Staubli VAL3: getMedian.pgx

public program getMedian(num& x_nInput[], num& x_nMedian)
  local num l_nCount
  local num l_nSmallsub
  local num l_nSort
  local num l_nTemp
begin

  // do a selection sort:
  // The idea of Selection Sort is that we repeatedly find the smallest element in the unsorted part of the array and swap it with the first element in the unsorted part of the array.

  resize(nTemp, 1, size(x_nInput))
  resize(nCopy, 1, size(x_nInput))

  for l_nCount = 0 to size(x_nInput)-1
    nCopy[l_nCount] = x_nInput[l_nCount]
  endFor


  for l_nCount = 0 to size(nCopy)-1
    l_nSmallsub = l_nCount

    for l_nSort = l_nCount+1 to size(nCopy)-1
      if nCopy[l_nSort] < nCopy[l_nSmallsub]
        l_nSmallsub = l_nSort
      endIf
    endFor

    l_nTemp = nCopy[l_nCount]
    nTemp[l_nCount] = nCopy[l_nSmallsub]
    nCopy[l_nSmallsub] = l_nTemp

  endFor

  if size(nCopy)%2 != 0
    // extract middle value of sorted list
    x_nMedian = nTemp[((size(nCopy)+1)/2)-1]
  else
    x_nMedian = (nTemp[(size(nCopy)/2)-1] + nTemp[size(nCopy)/2])/2
  endIf


end
